// TIA Portal V18 export
DATA_BLOCK "Machine infromation"   // DB80
{ S7_Optimized_Access := 'TRUE' }
VERSION : 0.1
// stored: AutoNumber true, DBAccessibleFromOPCUA true, IsOnlyStoredInLoadMemory false, IsRetainMemResEnabled false, IsWriteProtectedInAS false, MemoryReserve 100
   VAR RETAIN
      "Software No" : String := 'P-761.V0 20220930';
   END_VAR
BEGIN
END_DATA_BLOCK
